# EPICS substitutions: ecmcApp/Db/pmac.substitutions
file pmac.template {
pattern {P,     PORT,    ADDR, TIMEOUT }
{        IOC2:, MC_CPU1,    0,    1.0 }
}
